// TIA Portal V16 export
// export: Created 2022-04-18T16:31:02.3222711Z, ExportSetting WithDefaults, DisplayName Totally Integrated Automation Portal, DisplayVersion V16 Update 3, DisplayName TIA Portal Version Control Interface, DisplayVersion V16 Update 2, DisplayName TIA Portal Openness, DisplayVersion V16 Update 3, DisplayName STEP 7 Professional, DisplayVersion V16 Update 3, DisplayName STEP 7 Safety, DisplayVersion V16, DisplayName WinCC Professional, DisplayVersion V16 Update 3
TYPE "UT38151_Dy_SubTimeEventRTC"
TITLE = Dynamic UDT [SUBROUTINE] — Event Timer RTC
// PRACTICAL SERIES AUTOMATION LIBRARY (PAL)   —   COPYRIGHT 2020 – M. GLEDHILL (MIT LICENCE)
//                   ———— ◆ ————
// FULL ONLINE DOCUMENTATION IS AVAILABLE AT: https://practicalseries.com/2001-pal/index.html
// stored: IsFailsafeCompliant false
   STRUCT
      revInfo { ExternalWritable := 'False'} : "UT01000_St_SysRevision";   // ▀▀▀▀ UDT CURRENT REVISION
      ___________0010_0 { ExternalAccessible := 'False'; ExternalVisible := 'False'; ExternalWritable := 'False'} : Int;
      ___________0010_1 { ExternalAccessible := 'False'; ExternalVisible := 'False'; ExternalWritable := 'False'} : Int;   // ▀▀▀▀ STATUS SIGNALS
      status_Running { ExternalWritable := 'False'} : Bool;   // STATUS — Event timer is running (1 = running, 0 = stopped)
      ___________0020_0 { ExternalAccessible := 'False'; ExternalVisible := 'False'; ExternalWritable := 'False'} : Int;
      ___________0020_1 { ExternalAccessible := 'False'; ExternalVisible := 'False'; ExternalWritable := 'False'} : Int;   // ▀▀▀▀ EVENT TIMER RESULTS
      actual_StartTime { ExternalWritable := 'False'} : DTL;   // ACTUAL — Start time — RTC value on rising edge of trigger signal
      actual_EndTime { ExternalWritable := 'False'} : DTL;   // ACTUAL — End time — RTC value on falling edge of trigger signal
      actual_Duration { ExternalWritable := 'False'} : LTime;   // ACTUAL — Duration (end time - start time)
      actual_DurationSec { ExternalWritable := 'False'} : Real;   // ACTUAL — Duration (end time - start time) in seconds
   END_STRUCT;
   // revInfo.REV_BLOCK := 'UT38151';
   // revInfo.REV_NUMBER := '002.000';
   // revInfo.REV_DATE := '2022-04-16';
   // revInfo.REV_AUTHOR := 'M. Gledhill';
END_TYPE
